{attribute 'qualified_only'}
VAR_GLOBAL
	aTaskLogger			: ARRAY[1..SIZEOF(TwinCAT_SystemInfoVarList._TaskInfo)/SIZEOF(PlcTaskSystemInfo)] OF FB_Log4TcTask;
END_VAR

(* stored: Version 1.1.0.1, ProductVersion 3.1.4024.0
   GVL GlobalVariables: Id {aaa31d82-0afd-48ec-8faa-fd71178550ce} *)
